// Mitsubishi GX Works2 project: replay2   PLC: Q03UDV

PROGRAM MAIN
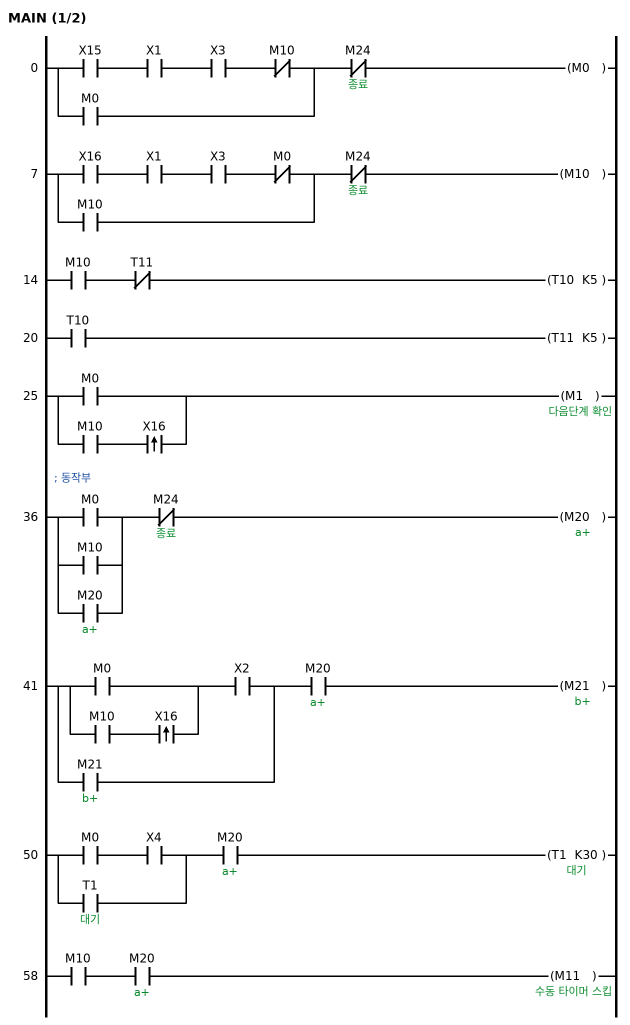
0     LD      X15
      AND     X1
      AND     X3
      ANI     M10
      OR      M0
      ANI     M24  ; 종료
      OUT     M0
7     LD      X16
      AND     X1
      AND     X3
      ANI     M0
      OR      M10
      ANI     M24  ; 종료
      OUT     M10
14    LD      M10
      ANI     T11
      OUT     T10 K5
20    LD      T10
      OUT     T11 K5
25    LD      M0
      LD      M10
      ANDP    X16
      ORB
      OUT     M1  ; 다음단계 확인
; 동작부
36    LD      M0
      OR      M10
      OR      M20  ; a+
      ANI     M24  ; 종료
      OUT     M20  ; a+
41    LD      M0
      LD      M10
      ANDP    X16
      ORB
      AND     X2
      OR      M21  ; b+
      AND     M20  ; a+
      OUT     M21  ; b+
50    LD      M0
      AND     X4
      OR      T1  ; 대기
      AND     M20  ; a+
      OUT     T1 K30  ; 대기
58    LD      M10
      AND     M20  ; a+
      OUT     M11  ; 수동 타이머 스킵
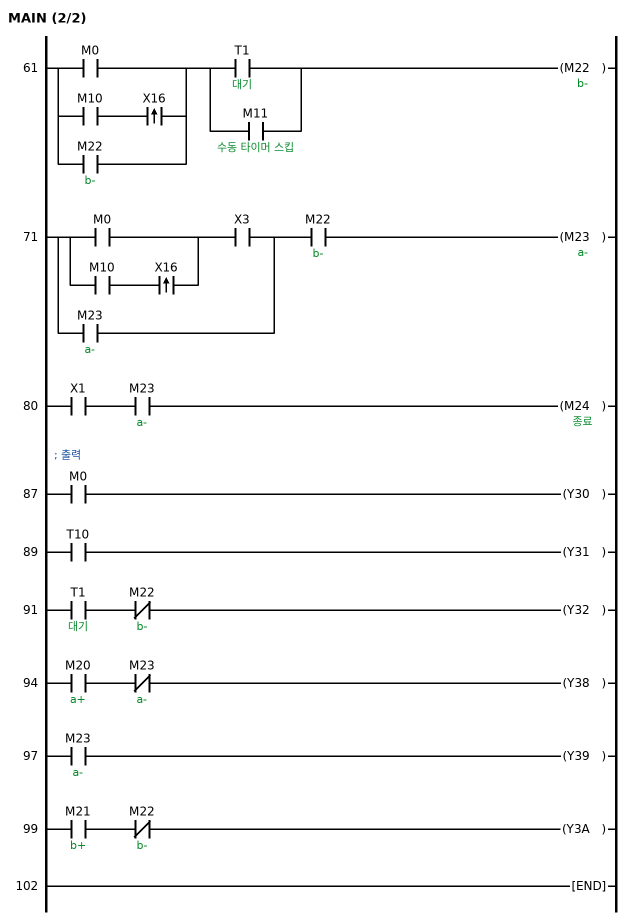
61    LD      M0
      LD      M10
      ANDP    X16
      ORB
      OR      M22  ; b-
      LD      T1  ; 대기
      OR      M11  ; 수동 타이머 스킵
      ANB
      OUT     M22  ; b-
71    LD      M0
      LD      M10
      ANDP    X16
      ORB
      AND     X3
      OR      M23  ; a-
      AND     M22  ; b-
      OUT     M23  ; a-
80    LD      X1
      AND     M23  ; a-
      OUT     M24  ; 종료
; 출력
87    LD      M0
      OUT     Y30
89    LD      T10
      OUT     Y31
91    LD      T1  ; 대기
      ANI     M22  ; b-
      OUT     Y32
94    LD      M20  ; a+
      ANI     M23  ; a-
      OUT     Y38
97    LD      M23  ; a-
      OUT     Y39
99    LD      M21  ; b+
      ANI     M22  ; b-
      OUT     Y3A
102   END
END_PROGRAM
